{attribute 'qualified_only'}
VAR_GLOBAL CONSTANT
	NumberOfWarningArea		: INT := 2;
END_VAR

(* stored: Version 1.1.0.1
   GVL Param: Id {c1bbae71-d283-4734-b7b1-71381b391320}, ParameterList True *)
